// TIA Portal V16 export
// export: Created 2025-10-06T17:54:28.7609427Z, ExportSetting WithDefaults, DisplayName Totally Integrated Automation Portal, DisplayVersion V16, DisplayName TIA Portal Version Control Interface, DisplayVersion V16, DisplayName TIA Portal Openness, DisplayVersion V16, DisplayName STEP 7 Professional, DisplayVersion V16, DisplayName STEP 7 Safety, DisplayVersion V16, DisplayName WinCC Advanced, DisplayVersion V16
FUNCTION "SafetyFunction_Block" : Void   // FC12, LAD
VERSION : 0.1
// stored: AutoNumber true, IsIECCheckEnabled false, UDAEnableTagReadback false
   VAR_INPUT
      "ESB NC Contact" : Bool;
      "ESB NO Contact" : Bool;
      "Reset NO Contact" : Bool;
      "SAFE door 1 NC Contact" : Bool;
      "SAFE door 2 NC Contact" : Bool;
      "Safety Relais NO Contact" : Bool;
   END_VAR
   VAR_OUTPUT
      SAFE_OK_Signal : Bool;
   END_VAR
BEGIN

REGION Network 1: +MC-21K6:1 - Noodstop Circuit
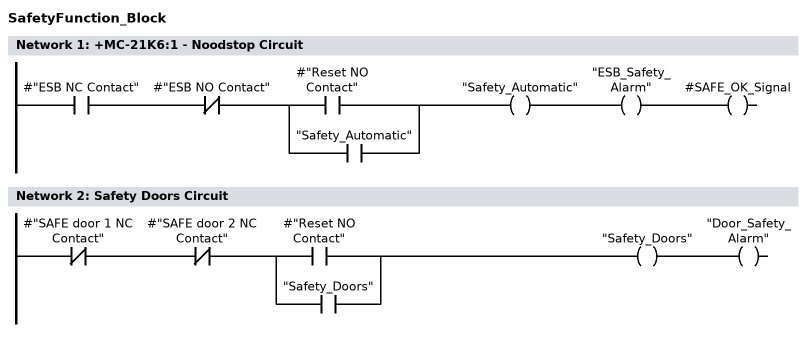
   RUNG wire#powerrail
      Contact( #"ESB NC Contact" )
      I_Contact( #"ESB NO Contact" )
      wire#w1
      Contact( #"Reset NO Contact" )
      wire#w2
      Coil( "Safety_Automatic" )
      Coil( "ESB_Safety_Alarm" )
      Coil( #SAFE_OK_Signal )
   END_RUNG
   RUNG wire#w1
      Contact( "Safety_Automatic" )
   END_RUNG wire#w2
   // the same network as SCL:
   "Safety_Automatic" := #"ESB NC Contact" AND NOT #"ESB NO Contact" AND (#"Reset NO Contact" OR "Safety_Automatic");
   "ESB_Safety_Alarm" := "Safety_Automatic";
   #SAFE_OK_Signal := "Safety_Automatic";
END_REGION

REGION Network 2: Safety Doors Circuit
   RUNG wire#powerrail
      I_Contact( #"SAFE door 1 NC Contact" )
      I_Contact( #"SAFE door 2 NC Contact" )
      wire#w1
      Contact( #"Reset NO Contact" )
      wire#w2
      Coil( "Safety_Doors" )
      Coil( "Door_Safety_Alarm" )
   END_RUNG
   RUNG wire#w1
      Contact( "Safety_Doors" )
   END_RUNG wire#w2
   // the same network as SCL:
   "Safety_Doors" := NOT #"SAFE door 1 NC Contact" AND NOT #"SAFE door 2 NC Contact" AND (#"Reset NO Contact" OR "Safety_Doors");
   "Door_Safety_Alarm" := "Safety_Doors";
END_REGION
END_FUNCTION
